% RSLogix 500 project Industrial_Bottle_Packaging_Line.RSS, saved by version 8.30.00.16 %
PROJECT "PROC1"    % processor: Bul.1763 MicroLogix 1100 Series B %

PROGRAM FILES
  LAD 2 "MAIN"  11 rungs
  LAD 3 "I / O"  27 rungs
  LAD 4 "MODE CTRL"  9 rungs
  LAD 5 "SNS IN CTR"  6 rungs
  LAD 6 "SIMULATION"  39 rungs
  LAD 7 "DEVICE CTR"  6 rungs
  LAD 8 "CYCLE RST"  2 rungs
  LAD 9 "HOURMETER"  8 rungs
  LAD 10 "ALARMS"  21 rungs

DATA FILES
  O0 OUTPUT  7 elements
  I1 INPUT  12 elements
  S2 STATUS  66 elements
  B3 BINARY  11 elements
  T4 TIMER  21 elements
  C5 COUNTER  1 elements
  R6 CONTROL  1 elements
  N7 INTEGER  23 elements
  F8 FLOAT  1 elements
  L9 LONGINT  1 elements

LADDER 2 "MAIN"
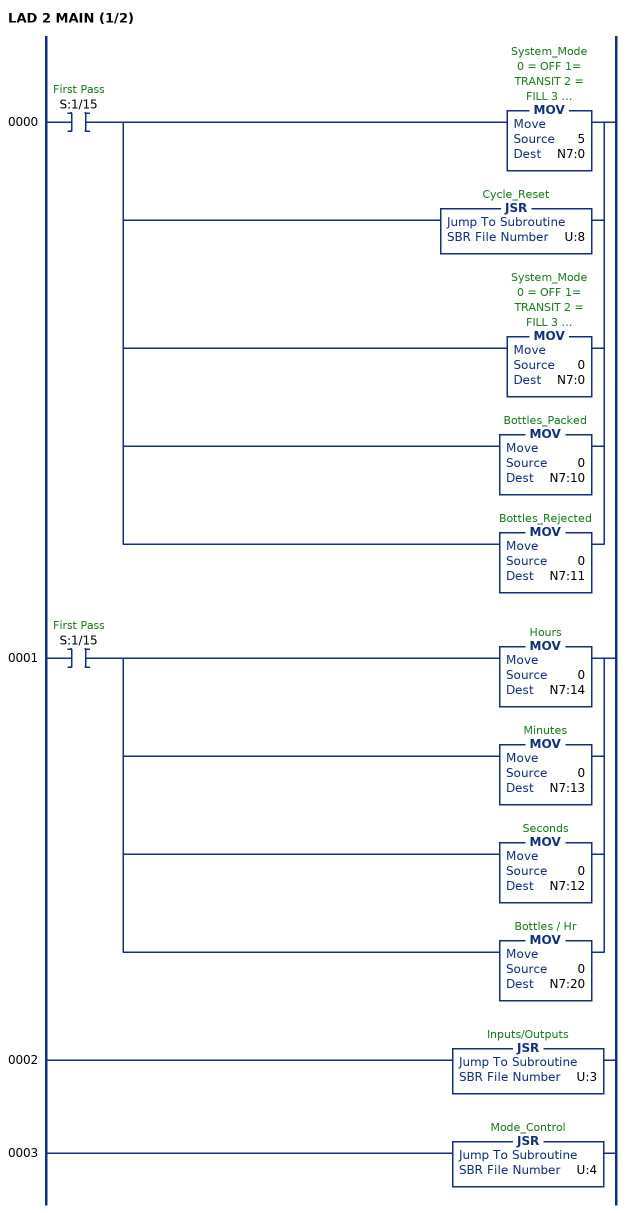
% Rung: 0 %
SOR XIC S:1/15 BST MOV 5 N7:0 NXB JSR U:8 NXB MOV 0 N7:0 NXB MOV 0 N7:10 NXB MOV 0 N7:11 BND EOR
%   S:1/15  "First Pass" %
%   N7:0  "System_Mode 0 = OFF 1= TRANSIT 2 = FILL 3 = CAPPING 4 = SORTING 5= CYC.R" %
%   U:8  "Cycle_Reset" %
%   N7:10  "Bottles_Packed" %
%   N7:11  "Bottles_Rejected" %
% Rung: 1 %
SOR XIC S:1/15 BST MOV 0 N7:14 NXB MOV 0 N7:13 NXB MOV 0 N7:12 NXB MOV 0 N7:20 BND EOR
%   S:1/15  "First Pass" %
%   N7:14  "Hours" %
%   N7:13  "Minutes" %
%   N7:12  "Seconds" %
%   N7:20  "Bottles / Hr" %
% Rung: 2 %
SOR JSR U:3 EOR
%   U:3  "Inputs/Outputs" %
% Rung: 3 %
SOR JSR U:4 EOR
%   U:4  "Mode_Control" %

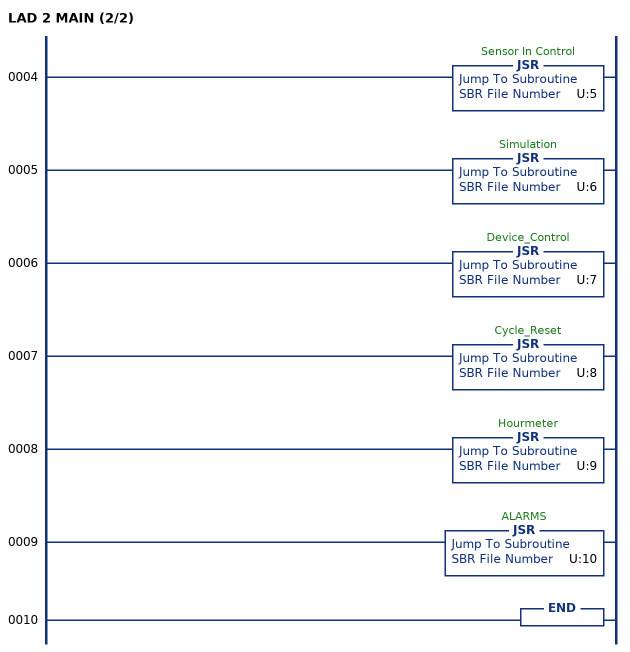
% Rung: 4 %
SOR JSR U:5 EOR
%   U:5  "Sensor In Control" %
% Rung: 5 %
SOR JSR U:6 EOR
%   U:6  "Simulation" %
% Rung: 6 %
SOR JSR U:7 EOR
%   U:7  "Device_Control" %
% Rung: 7 %
SOR JSR U:8 EOR
%   U:8  "Cycle_Reset" %
% Rung: 8 %
SOR JSR U:9 EOR
%   U:9  "Hourmeter" %
% Rung: 9 %
SOR JSR U:10 EOR
%   U:10  "ALARMS" %
% Rung: 10 %
SOR END EOR

LADDER 3 "I / O"
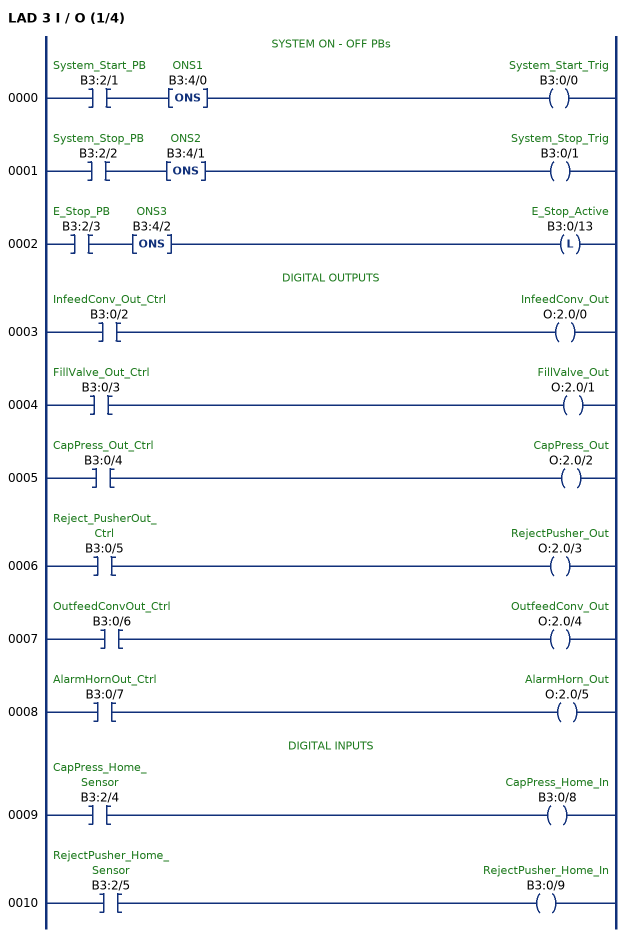
% Rung: 0 %
% SYSTEM ON - OFF PBs %
SOR XIC B3:2/1 ONS B3:4/0 OTE B3:0/0 EOR
%   B3:2/1  "System_Start_PB" %
%   B3:4/0  "ONS1" %
%   B3:0/0  "System_Start_Trig" %
% Rung: 1 %
SOR XIC B3:2/2 ONS B3:4/1 OTE B3:0/1 EOR
%   B3:2/2  "System_Stop_PB" %
%   B3:4/1  "ONS2" %
%   B3:0/1  "System_Stop_Trig" %
% Rung: 2 %
SOR XIC B3:2/3 ONS B3:4/2 OTL B3:0/13 EOR
%   B3:2/3  "E_Stop_PB" %
%   B3:4/2  "ONS3" %
%   B3:0/13  "E_Stop_Active" %
% Rung: 3 %
% DIGITAL OUTPUTS %
SOR XIC B3:0/2 OTE O:2.0/0 EOR
%   B3:0/2  "InfeedConv_Out_Ctrl" %
%   O:2.0/0  "InfeedConv_Out" %
% Rung: 4 %
SOR XIC B3:0/3 OTE O:2.0/1 EOR
%   B3:0/3  "FillValve_Out_Ctrl" %
%   O:2.0/1  "FillValve_Out" %
% Rung: 5 %
SOR XIC B3:0/4 OTE O:2.0/2 EOR
%   B3:0/4  "CapPress_Out_Ctrl" %
%   O:2.0/2  "CapPress_Out" %
% Rung: 6 %
SOR XIC B3:0/5 OTE O:2.0/3 EOR
%   B3:0/5  "Reject_PusherOut_ Ctrl" %
%   O:2.0/3  "RejectPusher_Out" %
% Rung: 7 %
SOR XIC B3:0/6 OTE O:2.0/4 EOR
%   B3:0/6  "OutfeedConvOut_Ctrl" %
%   O:2.0/4  "OutfeedConv_Out" %
% Rung: 8 %
SOR XIC B3:0/7 OTE O:2.0/5 EOR
%   B3:0/7  "AlarmHornOut_Ctrl" %
%   O:2.0/5  "AlarmHorn_Out" %
% Rung: 9 %
% DIGITAL INPUTS %
SOR XIC B3:2/4 OTE B3:0/8 EOR
%   B3:2/4  "CapPress_Home_Sensor" %
%   B3:0/8  "CapPress_Home_In" %
% Rung: 10 %
SOR XIC B3:2/5 OTE B3:0/9 EOR
%   B3:2/5  "RejectPusher_Home_ Sensor" %
%   B3:0/9  "RejectPusher_Home_In" %

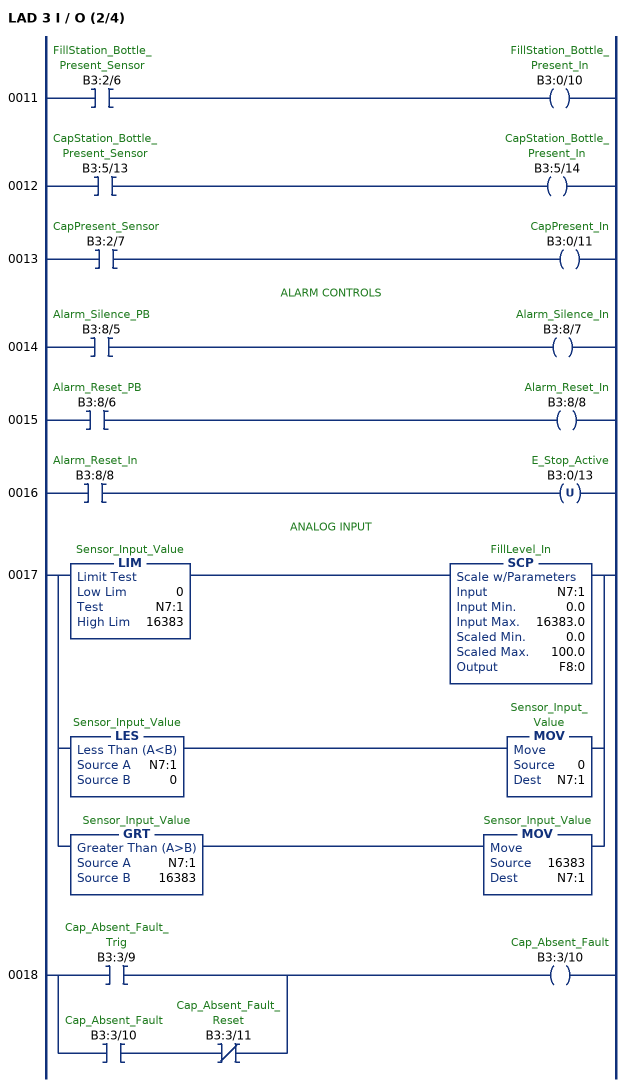
% Rung: 11 %
SOR XIC B3:2/6 OTE B3:0/10 EOR
%   B3:2/6  "FillStation_Bottle_ Present_Sensor" %
%   B3:0/10  "FillStation_Bottle_ Present_In" %
% Rung: 12 %
SOR XIC B3:5/13 OTE B3:5/14 EOR
%   B3:5/13  "CapStation_Bottle_ Present_Sensor" %
%   B3:5/14  "CapStation_Bottle_ Present_In" %
% Rung: 13 %
SOR XIC B3:2/7 OTE B3:0/11 EOR
%   B3:2/7  "CapPresent_Sensor" %
%   B3:0/11  "CapPresent_In" %
% Rung: 14 %
% ALARM CONTROLS %
SOR XIC B3:8/5 OTE B3:8/7 EOR
%   B3:8/5  "Alarm_Silence_PB" %
%   B3:8/7  "Alarm_Silence_In" %
% Rung: 15 %
SOR XIC B3:8/6 OTE B3:8/8 EOR
%   B3:8/6  "Alarm_Reset_PB" %
%   B3:8/8  "Alarm_Reset_In" %
% Rung: 16 %
SOR XIC B3:8/8 OTU B3:0/13 EOR
%   B3:8/8  "Alarm_Reset_In" %
%   B3:0/13  "E_Stop_Active" %
% Rung: 17 %
% ANALOG INPUT %
SOR BST LIM 0 N7:1 16383 SCP N7:1 0.0 16383.0 0.0 100.0 F8:0 NXB LES N7:1 0 MOV 0 N7:1 NXB GRT N7:1 16383 MOV 16383 N7:1 BND EOR
%   N7:1  "Sensor_Input_Value" %
%   F8:0  "FillLevel_In" %
% Rung: 18 %
SOR BST XIC B3:3/9 NXB XIC B3:3/10 XIO B3:3/11 BND OTE B3:3/10 EOR
%   B3:3/9  "Cap_Absent_Fault_ Trig" %
%   B3:3/10  "Cap_Absent_Fault" %
%   B3:3/11  "Cap_Absent_Fault_ Reset" %

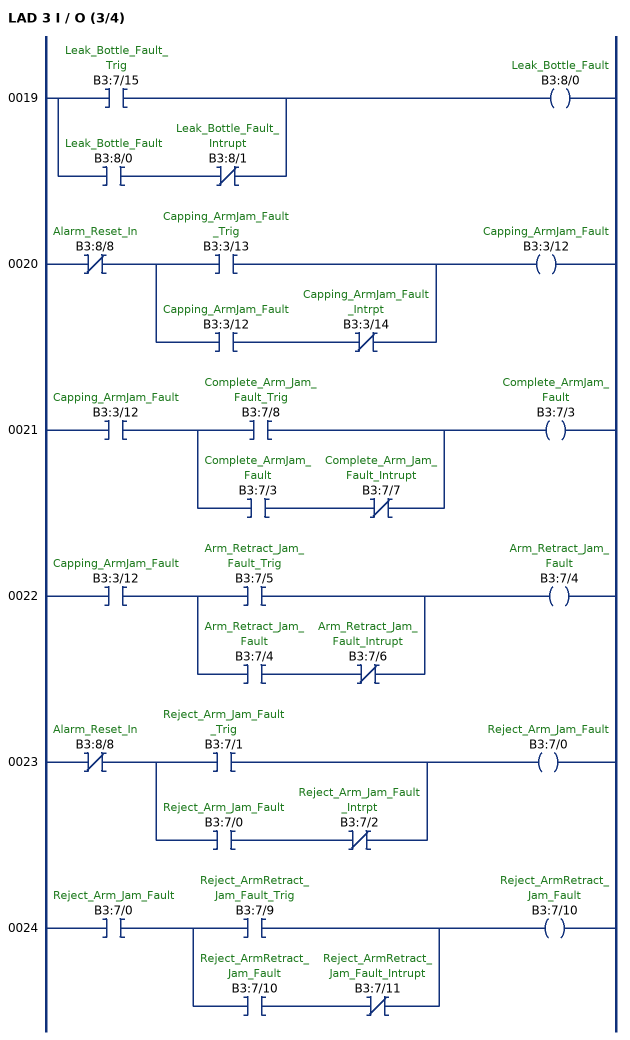
% Rung: 19 %
SOR BST XIC B3:7/15 NXB XIC B3:8/0 XIO B3:8/1 BND OTE B3:8/0 EOR
%   B3:7/15  "Leak_Bottle_Fault_ Trig" %
%   B3:8/0  "Leak_Bottle_Fault" %
%   B3:8/1  "Leak_Bottle_Fault_ Intrupt" %
% Rung: 20 %
SOR XIO B3:8/8 BST XIC B3:3/13 NXB XIC B3:3/12 XIO B3:3/14 BND OTE B3:3/12 EOR
%   B3:8/8  "Alarm_Reset_In" %
%   B3:3/13  "Capping_ArmJam_Fault _Trig" %
%   B3:3/12  "Capping_ArmJam_Fault" %
%   B3:3/14  "Capping_ArmJam_Fault _Intrpt" %
% Rung: 21 %
SOR XIC B3:3/12 BST XIC B3:7/8 NXB XIC B3:7/3 XIO B3:7/7 BND OTE B3:7/3 EOR
%   B3:3/12  "Capping_ArmJam_Fault" %
%   B3:7/8  "Complete_Arm_Jam_ Fault_Trig" %
%   B3:7/3  "Complete_ArmJam_ Fault" %
%   B3:7/7  "Complete_Arm_Jam_ Fault_Intrupt" %
% Rung: 22 %
SOR XIC B3:3/12 BST XIC B3:7/5 NXB XIC B3:7/4 XIO B3:7/6 BND OTE B3:7/4 EOR
%   B3:3/12  "Capping_ArmJam_Fault" %
%   B3:7/5  "Arm_Retract_Jam_ Fault_Trig" %
%   B3:7/4  "Arm_Retract_Jam_ Fault" %
%   B3:7/6  "Arm_Retract_Jam_ Fault_Intrupt" %
% Rung: 23 %
SOR XIO B3:8/8 BST XIC B3:7/1 NXB XIC B3:7/0 XIO B3:7/2 BND OTE B3:7/0 EOR
%   B3:8/8  "Alarm_Reset_In" %
%   B3:7/1  "Reject_Arm_Jam_Fault _Trig" %
%   B3:7/0  "Reject_Arm_Jam_Fault" %
%   B3:7/2  "Reject_Arm_Jam_Fault _Intrpt" %
% Rung: 24 %
SOR XIC B3:7/0 BST XIC B3:7/9 NXB XIC B3:7/10 XIO B3:7/11 BND OTE B3:7/10 EOR
%   B3:7/0  "Reject_Arm_Jam_Fault" %
%   B3:7/9  "Reject_ArmRetract_ Jam_Fault_Trig" %
%   B3:7/10  "Reject_ArmRetract_ Jam_Fault" %
%   B3:7/11  "Reject_ArmRetract_ Jam_Fault_Intrupt" %

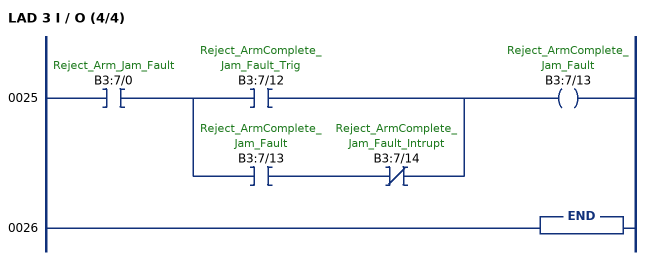
% Rung: 25 %
SOR XIC B3:7/0 BST XIC B3:7/12 NXB XIC B3:7/13 XIO B3:7/14 BND OTE B3:7/13 EOR
%   B3:7/0  "Reject_Arm_Jam_Fault" %
%   B3:7/12  "Reject_ArmComplete_ Jam_Fault_Trig" %
%   B3:7/13  "Reject_ArmComplete_ Jam_Fault" %
%   B3:7/14  "Reject_ArmComplete_ Jam_Fault_Intrupt" %
% Rung: 26 %
SOR END EOR

LADDER 4 "MODE CTRL"
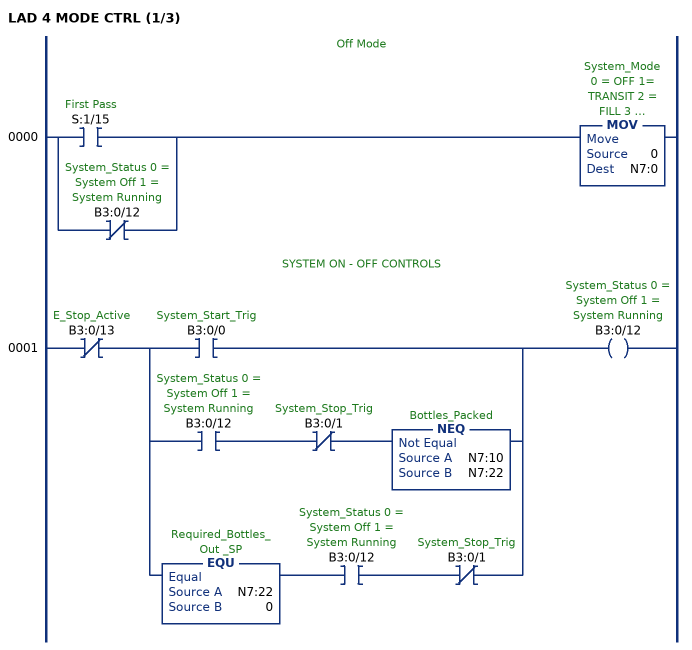
% Rung: 0 %
% Off Mode %
SOR BST XIC S:1/15 NXB XIO B3:0/12 BND MOV 0 N7:0 EOR
%   S:1/15  "First Pass" %
%   B3:0/12  "System_Status 0 = System Off 1 = System Running" %
%   N7:0  "System_Mode 0 = OFF 1= TRANSIT 2 = FILL 3 = CAPPING 4 = SORTING 5= CYC.R" %
% Rung: 1 %
% SYSTEM ON - OFF CONTROLS %
SOR XIO B3:0/13 BST XIC B3:0/0 NXB XIC B3:0/12 XIO B3:0/1 NEQ N7:10 N7:22 NXB EQU N7:22 0 XIC B3:0/12 XIO B3:0/1 BND OTE B3:0/12 EOR
%   B3:0/13  "E_Stop_Active" %
%   B3:0/0  "System_Start_Trig" %
%   B3:0/12  "System_Status 0 = System Off 1 = System Running" %
%   B3:0/1  "System_Stop_Trig" %
%   N7:10  "Bottles_Packed" %
%   N7:22  "Required_Bottles_Out _SP" %

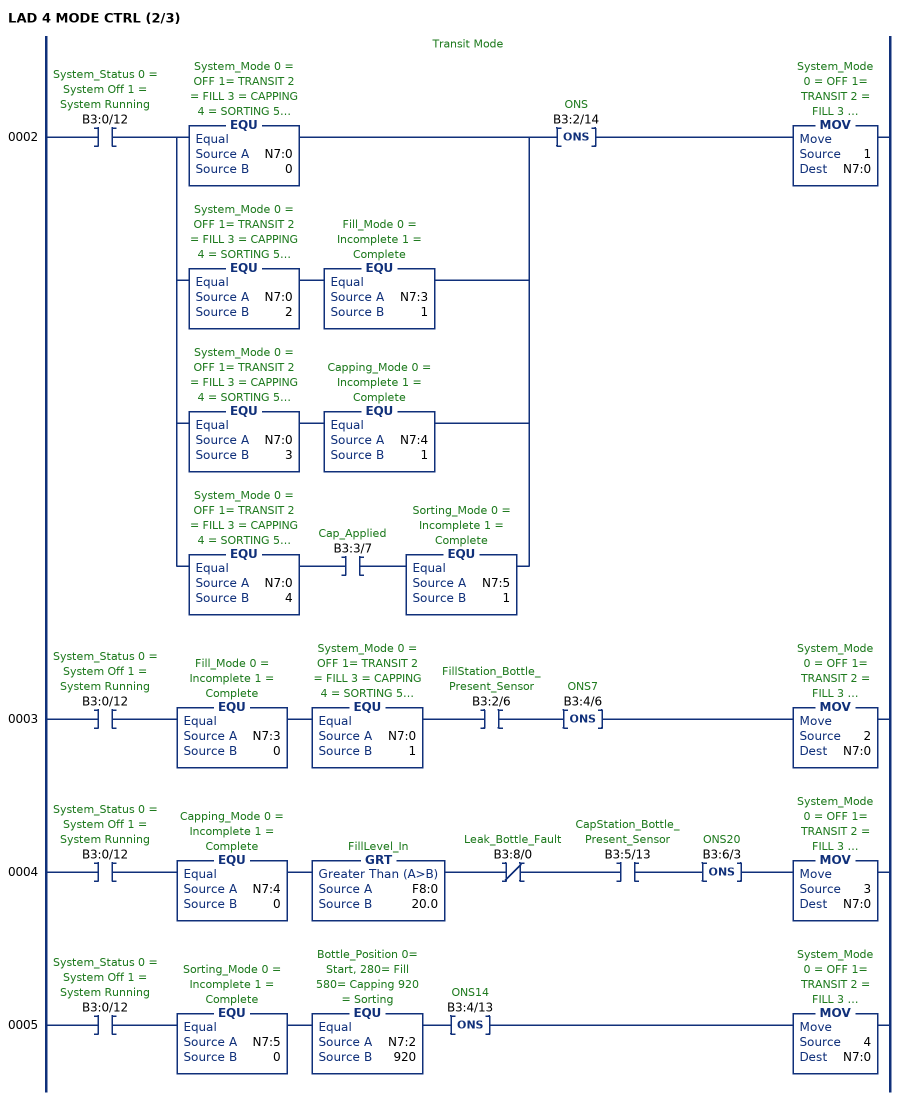
% Rung: 2 %
% Transit Mode %
SOR XIC B3:0/12 BST EQU N7:0 0 NXB EQU N7:0 2 EQU N7:3 1 NXB EQU N7:0 3 EQU N7:4 1 NXB EQU N7:0 4 XIC B3:3/7 EQU N7:5 1 BND ONS B3:2/14 MOV 1 N7:0 EOR
%   B3:0/12  "System_Status 0 = System Off 1 = System Running" %
%   N7:0  "System_Mode 0 = OFF 1= TRANSIT 2 = FILL 3 = CAPPING 4 = SORTING 5= CYC.R" %
%   N7:3  "Fill_Mode 0 = Incomplete 1 = Complete" %
%   N7:4  "Capping_Mode 0 = Incomplete 1 = Complete" %
%   B3:3/7  "Cap_Applied" %
%   N7:5  "Sorting_Mode 0 = Incomplete 1 = Complete" %
%   B3:2/14  "ONS" %
% Rung: 3 %
SOR XIC B3:0/12 EQU N7:3 0 EQU N7:0 1 XIC B3:2/6 ONS B3:4/6 MOV 2 N7:0 EOR
%   B3:0/12  "System_Status 0 = System Off 1 = System Running" %
%   N7:3  "Fill_Mode 0 = Incomplete 1 = Complete" %
%   N7:0  "System_Mode 0 = OFF 1= TRANSIT 2 = FILL 3 = CAPPING 4 = SORTING 5= CYC.R" %
%   B3:2/6  "FillStation_Bottle_ Present_Sensor" %
%   B3:4/6  "ONS7" %
% Rung: 4 %
SOR XIC B3:0/12 EQU N7:4 0 GRT F8:0 20.0 XIO B3:8/0 XIC B3:5/13 ONS B3:6/3 MOV 3 N7:0 EOR
%   B3:0/12  "System_Status 0 = System Off 1 = System Running" %
%   N7:4  "Capping_Mode 0 = Incomplete 1 = Complete" %
%   F8:0  "FillLevel_In" %
%   B3:8/0  "Leak_Bottle_Fault" %
%   B3:5/13  "CapStation_Bottle_ Present_Sensor" %
%   B3:6/3  "ONS20" %
%   N7:0  "System_Mode 0 = OFF 1= TRANSIT 2 = FILL 3 = CAPPING 4 = SORTING 5= CYC.R" %
% Rung: 5 %
SOR XIC B3:0/12 EQU N7:5 0 EQU N7:2 920 ONS B3:4/13 MOV 4 N7:0 EOR
%   B3:0/12  "System_Status 0 = System Off 1 = System Running" %
%   N7:5  "Sorting_Mode 0 = Incomplete 1 = Complete" %
%   N7:2  "Bottle_Position 0= Start, 280= Fill 580= Capping 920 = Sorting" %
%   B3:4/13  "ONS14" %
%   N7:0  "System_Mode 0 = OFF 1= TRANSIT 2 = FILL 3 = CAPPING 4 = SORTING 5= CYC.R" %

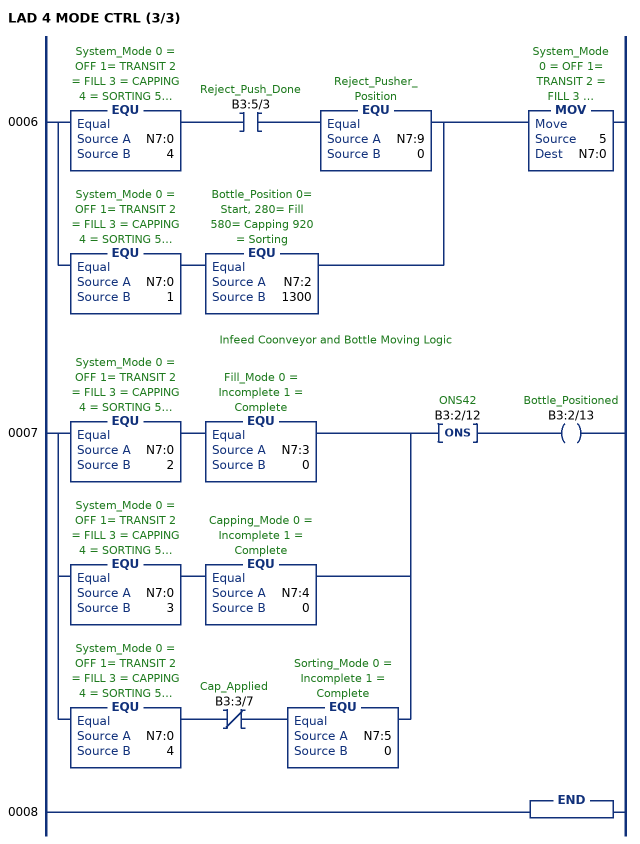
% Rung: 6 %
SOR BST EQU N7:0 4 XIC B3:5/3 EQU N7:9 0 NXB EQU N7:0 1 EQU N7:2 1300 BND MOV 5 N7:0 EOR
%   N7:0  "System_Mode 0 = OFF 1= TRANSIT 2 = FILL 3 = CAPPING 4 = SORTING 5= CYC.R" %
%   B3:5/3  "Reject_Push_Done" %
%   N7:9  "Reject_Pusher_ Position" %
%   N7:2  "Bottle_Position 0= Start, 280= Fill 580= Capping 920 = Sorting" %
% Rung: 7 %
% Infeed Coonveyor and Bottle Moving Logic %
SOR BST EQU N7:0 2 EQU N7:3 0 NXB EQU N7:0 3 EQU N7:4 0 NXB EQU N7:0 4 XIO B3:3/7 EQU N7:5 0 BND ONS B3:2/12 OTE B3:2/13 EOR
%   N7:0  "System_Mode 0 = OFF 1= TRANSIT 2 = FILL 3 = CAPPING 4 = SORTING 5= CYC.R" %
%   N7:3  "Fill_Mode 0 = Incomplete 1 = Complete" %
%   N7:4  "Capping_Mode 0 = Incomplete 1 = Complete" %
%   B3:3/7  "Cap_Applied" %
%   N7:5  "Sorting_Mode 0 = Incomplete 1 = Complete" %
%   B3:2/12  "ONS42" %
%   B3:2/13  "Bottle_Positioned" %
% Rung: 8 %
SOR END EOR

LADDER 5 "SNS IN CTR"
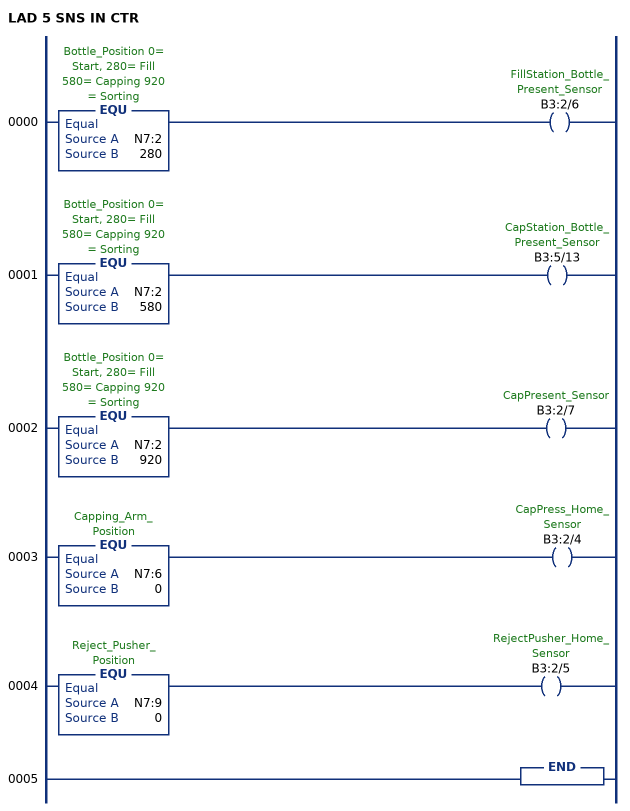
% Rung: 0 %
SOR EQU N7:2 280 OTE B3:2/6 EOR
%   N7:2  "Bottle_Position 0= Start, 280= Fill 580= Capping 920 = Sorting" %
%   B3:2/6  "FillStation_Bottle_ Present_Sensor" %
% Rung: 1 %
SOR EQU N7:2 580 OTE B3:5/13 EOR
%   N7:2  "Bottle_Position 0= Start, 280= Fill 580= Capping 920 = Sorting" %
%   B3:5/13  "CapStation_Bottle_ Present_Sensor" %
% Rung: 2 %
SOR EQU N7:2 920 OTE B3:2/7 EOR
%   N7:2  "Bottle_Position 0= Start, 280= Fill 580= Capping 920 = Sorting" %
%   B3:2/7  "CapPresent_Sensor" %
% Rung: 3 %
SOR EQU N7:6 0 OTE B3:2/4 EOR
%   N7:6  "Capping_Arm_Position" %
%   B3:2/4  "CapPress_Home_Sensor" %
% Rung: 4 %
SOR EQU N7:9 0 OTE B3:2/5 EOR
%   N7:9  "Reject_Pusher_ Position" %
%   B3:2/5  "RejectPusher_Home_ Sensor" %
% Rung: 5 %
SOR END EOR

LADDER 6 "SIMULATION"
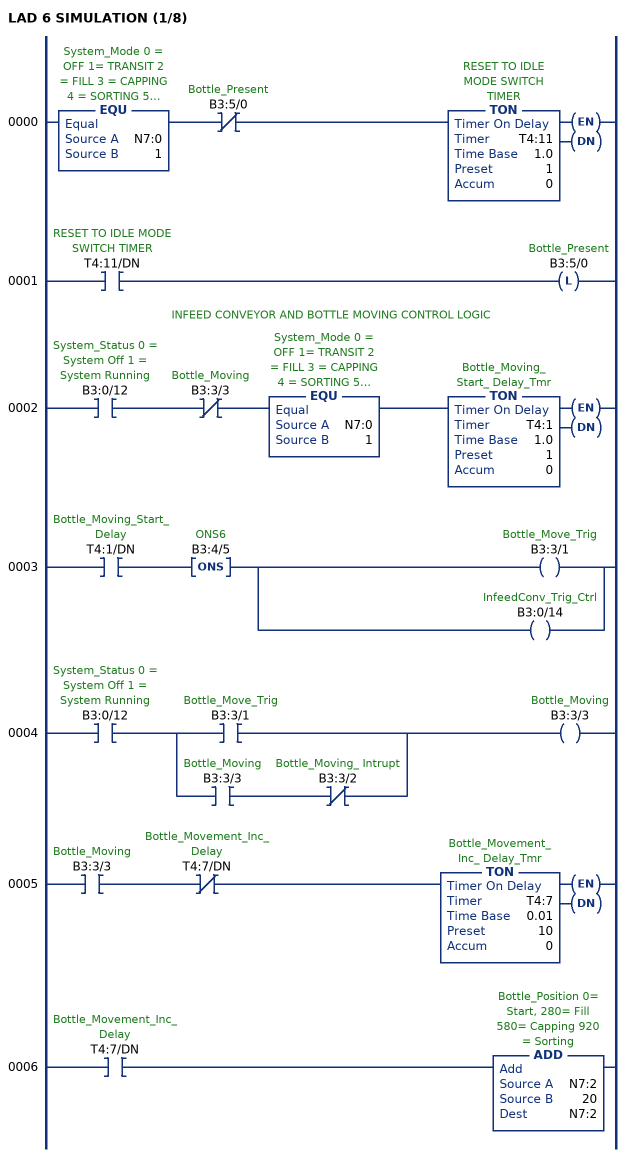
% Rung: 0 %
SOR EQU N7:0 1 XIO B3:5/0 TON T4:11 1.0 1 0 EOR
%   N7:0  "System_Mode 0 = OFF 1= TRANSIT 2 = FILL 3 = CAPPING 4 = SORTING 5= CYC.R" %
%   B3:5/0  "Bottle_Present" %
%   T4:11  "RESET TO IDLE MODE SWITCH TIMER" %
% Rung: 1 %
SOR XIC T4:11/DN OTL B3:5/0 EOR
%   T4:11  "RESET TO IDLE MODE SWITCH TIMER" %
%   B3:5/0  "Bottle_Present" %
% Rung: 2 %
% INFEED CONVEYOR AND BOTTLE MOVING CONTROL LOGIC %
SOR XIC B3:0/12 XIO B3:3/3 EQU N7:0 1 TON T4:1 1.0 1 0 EOR
%   B3:0/12  "System_Status 0 = System Off 1 = System Running" %
%   B3:3/3  "Bottle_Moving" %
%   N7:0  "System_Mode 0 = OFF 1= TRANSIT 2 = FILL 3 = CAPPING 4 = SORTING 5= CYC.R" %
%   T4:1  "Bottle_Moving_Start_ Delay_Tmr" %
% Rung: 3 %
SOR XIC T4:1/DN ONS B3:4/5 BST OTE B3:3/1 NXB OTE B3:0/14 BND EOR
%   T4:1/DN  "Bottle_Moving_Start_ Delay" %
%   B3:4/5  "ONS6" %
%   B3:3/1  "Bottle_Move_Trig" %
%   B3:0/14  "InfeedConv_Trig_Ctrl" %
% Rung: 4 %
SOR XIC B3:0/12 BST XIC B3:3/1 NXB XIC B3:3/3 XIO B3:3/2 BND OTE B3:3/3 EOR
%   B3:0/12  "System_Status 0 = System Off 1 = System Running" %
%   B3:3/1  "Bottle_Move_Trig" %
%   B3:3/3  "Bottle_Moving" %
%   B3:3/2  "Bottle_Moving_ Intrupt" %
% Rung: 5 %
SOR XIC B3:3/3 XIO T4:7/DN TON T4:7 0.01 10 0 EOR
%   B3:3/3  "Bottle_Moving" %
%   T4:7/DN  "Bottle_Movement_Inc_ Delay" %
%   T4:7  "Bottle_Movement_Inc_ Delay_Tmr" %
% Rung: 6 %
SOR XIC T4:7/DN ADD N7:2 20 N7:2 EOR
%   T4:7/DN  "Bottle_Movement_Inc_ Delay" %
%   N7:2  "Bottle_Position 0= Start, 280= Fill 580= Capping 920 = Sorting" %

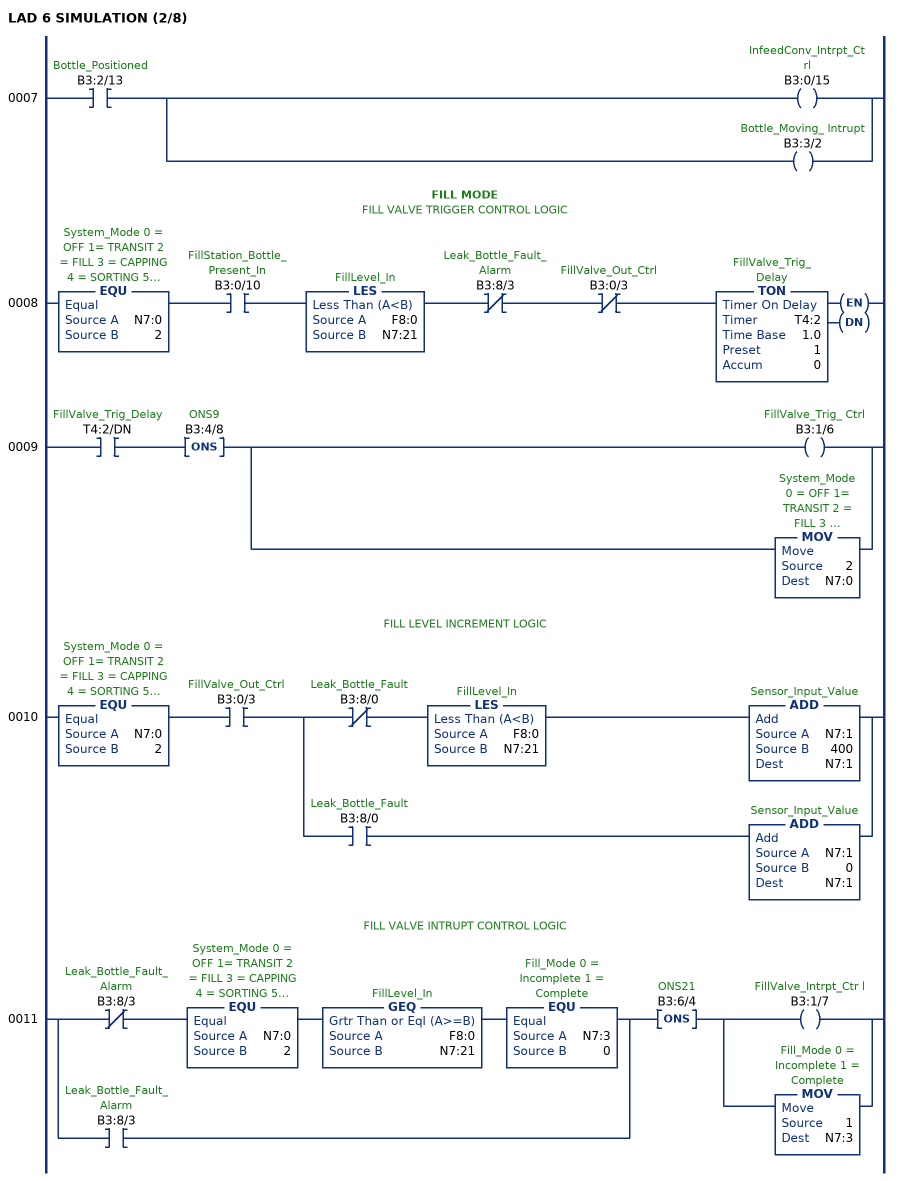
% Rung: 7 %
SOR XIC B3:2/13 BST OTE B3:0/15 NXB OTE B3:3/2 BND EOR
%   B3:2/13  "Bottle_Positioned" %
%   B3:0/15  "InfeedConv_Intrpt_Ct rl" %
%   B3:3/2  "Bottle_Moving_ Intrupt" %
% Rung: 8 %
% TITLE: FILL MODE %
% FILL VALVE TRIGGER CONTROL LOGIC %
SOR EQU N7:0 2 XIC B3:0/10 LES F8:0 N7:21 XIO B3:8/3 XIO B3:0/3 TON T4:2 1.0 1 0 EOR
%   N7:0  "System_Mode 0 = OFF 1= TRANSIT 2 = FILL 3 = CAPPING 4 = SORTING 5= CYC.R" %
%   B3:0/10  "FillStation_Bottle_ Present_In" %
%   F8:0  "FillLevel_In" %
%   N7:21  "Fill_LVL_SP" %
%   B3:8/3  "Leak_Bottle_Fault_ Alarm" %
%   B3:0/3  "FillValve_Out_Ctrl" %
%   T4:2  "FillValve_Trig_ Delay" %
% Rung: 9 %
SOR XIC T4:2/DN ONS B3:4/8 BST OTE B3:1/6 NXB MOV 2 N7:0 BND EOR
%   T4:2/DN  "FillValve_Trig_Delay" %
%   B3:4/8  "ONS9" %
%   B3:1/6  "FillValve_Trig_ Ctrl" %
%   N7:0  "System_Mode 0 = OFF 1= TRANSIT 2 = FILL 3 = CAPPING 4 = SORTING 5= CYC.R" %
% Rung: 10 %
% FILL LEVEL INCREMENT LOGIC %
SOR EQU N7:0 2 XIC B3:0/3 BST XIO B3:8/0 LES F8:0 N7:21 ADD N7:1 400 N7:1 NXB XIC B3:8/0 ADD N7:1 0 N7:1 BND EOR
%   N7:0  "System_Mode 0 = OFF 1= TRANSIT 2 = FILL 3 = CAPPING 4 = SORTING 5= CYC.R" %
%   B3:0/3  "FillValve_Out_Ctrl" %
%   B3:8/0  "Leak_Bottle_Fault" %
%   F8:0  "FillLevel_In" %
%   N7:21  "Fill_LVL_SP" %
%   N7:1  "Sensor_Input_Value" %
% Rung: 11 %
% FILL VALVE INTRUPT CONTROL LOGIC %
SOR BST XIO B3:8/3 EQU N7:0 2 GEQ F8:0 N7:21 EQU N7:3 0 NXB XIC B3:8/3 BND ONS B3:6/4 BST OTE B3:1/7 NXB MOV 1 N7:3 BND EOR
%   B3:8/3  "Leak_Bottle_Fault_ Alarm" %
%   N7:0  "System_Mode 0 = OFF 1= TRANSIT 2 = FILL 3 = CAPPING 4 = SORTING 5= CYC.R" %
%   F8:0  "FillLevel_In" %
%   N7:21  "Fill_LVL_SP" %
%   N7:3  "Fill_Mode 0 = Incomplete 1 = Complete" %
%   B3:6/4  "ONS21" %
%   B3:1/7  "FillValve_Intrpt_Ctr l" %

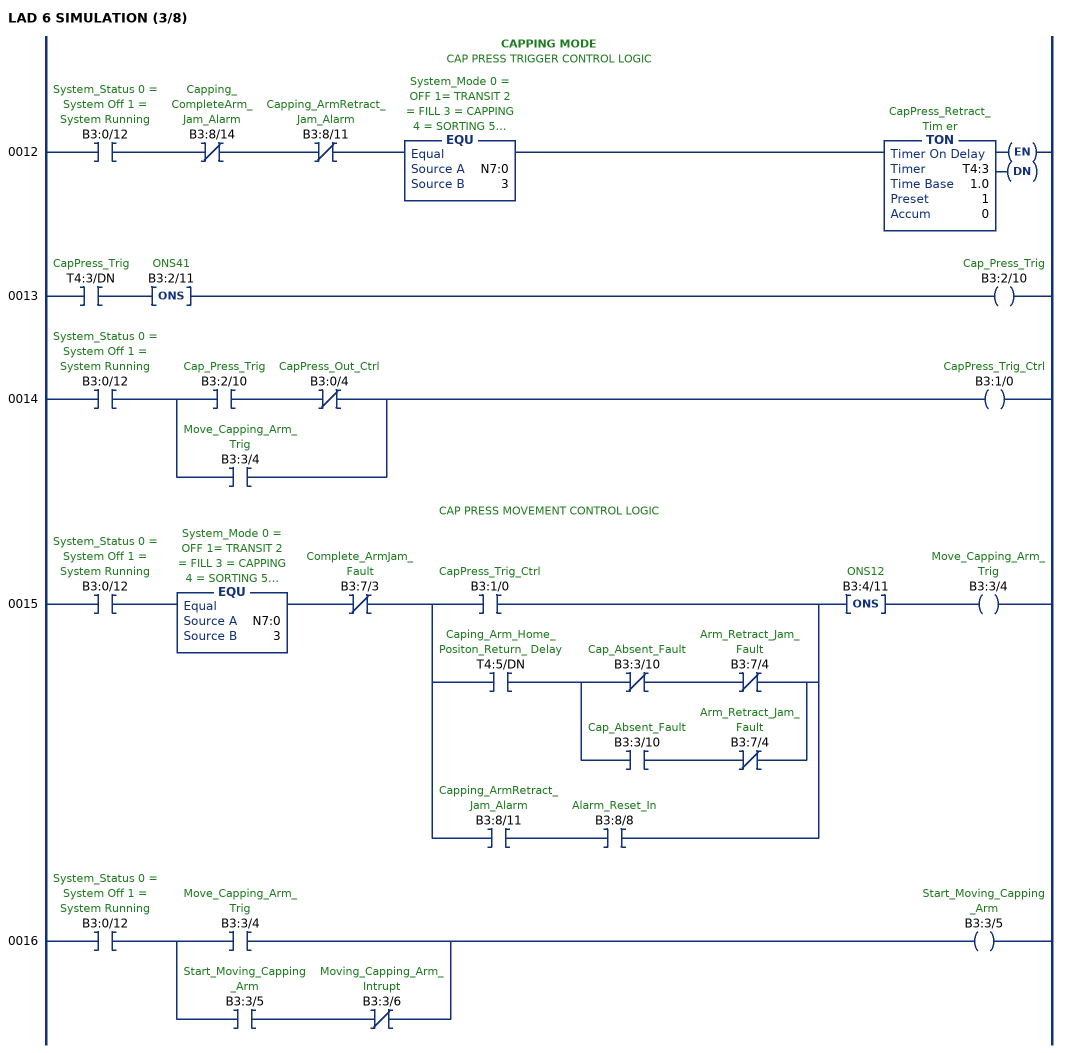
% Rung: 12 %
% TITLE: CAPPING MODE %
% CAP PRESS TRIGGER CONTROL LOGIC %
SOR XIC B3:0/12 XIO B3:8/14 XIO B3:8/11 EQU N7:0 3 TON T4:3 1.0 1 0 EOR
%   B3:0/12  "System_Status 0 = System Off 1 = System Running" %
%   B3:8/14  "Capping_CompleteArm_ Jam_Alarm" %
%   B3:8/11  "Capping_ArmRetract_ Jam_Alarm" %
%   N7:0  "System_Mode 0 = OFF 1= TRANSIT 2 = FILL 3 = CAPPING 4 = SORTING 5= CYC.R" %
%   T4:3  "CapPress_Retract_Tim er" %
% Rung: 13 %
SOR XIC T4:3/DN ONS B3:2/11 OTE B3:2/10 EOR
%   T4:3/DN  "CapPress_Trig" %
%   B3:2/11  "ONS41" %
%   B3:2/10  "Cap_Press_Trig" %
% Rung: 14 %
SOR XIC B3:0/12 BST XIC B3:2/10 XIO B3:0/4 NXB XIC B3:3/4 BND OTE B3:1/0 EOR
%   B3:0/12  "System_Status 0 = System Off 1 = System Running" %
%   B3:2/10  "Cap_Press_Trig" %
%   B3:0/4  "CapPress_Out_Ctrl" %
%   B3:3/4  "Move_Capping_Arm_ Trig" %
%   B3:1/0  "CapPress_Trig_Ctrl" %
% Rung: 15 %
% CAP PRESS MOVEMENT CONTROL LOGIC %
SOR XIC B3:0/12 EQU N7:0 3 XIO B3:7/3 BST XIC B3:1/0 NXB XIC T4:5/DN BST XIO B3:3/10 XIO B3:7/4 NXB XIC B3:3/10 XIO B3:7/4 BND NXB XIC B3:8/11 XIC B3:8/8 BND ONS B3:4/11 OTE B3:3/4 EOR
%   B3:0/12  "System_Status 0 = System Off 1 = System Running" %
%   N7:0  "System_Mode 0 = OFF 1= TRANSIT 2 = FILL 3 = CAPPING 4 = SORTING 5= CYC.R" %
%   B3:7/3  "Complete_ArmJam_ Fault" %
%   B3:1/0  "CapPress_Trig_Ctrl" %
%   T4:5/DN  "Caping_Arm_Home_ Positon_Return_ Delay" %
%   B3:3/10  "Cap_Absent_Fault" %
%   B3:7/4  "Arm_Retract_Jam_ Fault" %
%   B3:8/11  "Capping_ArmRetract_ Jam_Alarm" %
%   B3:8/8  "Alarm_Reset_In" %
%   B3:4/11  "ONS12" %
%   B3:3/4  "Move_Capping_Arm_ Trig" %
% Rung: 16 %
SOR XIC B3:0/12 BST XIC B3:3/4 NXB XIC B3:3/5 XIO B3:3/6 BND OTE B3:3/5 EOR
%   B3:0/12  "System_Status 0 = System Off 1 = System Running" %
%   B3:3/4  "Move_Capping_Arm_ Trig" %
%   B3:3/5  "Start_Moving_Capping _Arm" %
%   B3:3/6  "Moving_Capping_Arm_ Intrupt" %

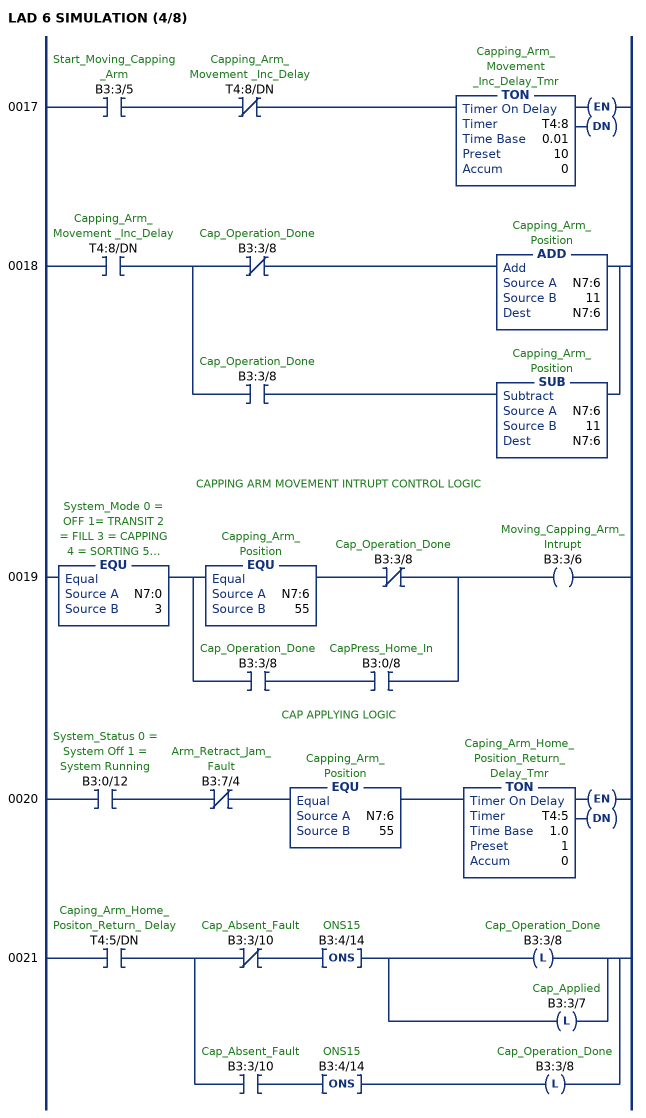
% Rung: 17 %
SOR XIC B3:3/5 XIO T4:8/DN TON T4:8 0.01 10 0 EOR
%   B3:3/5  "Start_Moving_Capping _Arm" %
%   T4:8/DN  "Capping_Arm_Movement _Inc_Delay" %
%   T4:8  "Capping_Arm_Movement _Inc_Delay_Tmr" %
% Rung: 18 %
SOR XIC T4:8/DN BST XIO B3:3/8 ADD N7:6 11 N7:6 NXB XIC B3:3/8 SUB N7:6 11 N7:6 BND EOR
%   T4:8/DN  "Capping_Arm_Movement _Inc_Delay" %
%   B3:3/8  "Cap_Operation_Done" %
%   N7:6  "Capping_Arm_Position" %
% Rung: 19 %
% CAPPING ARM MOVEMENT INTRUPT CONTROL LOGIC %
SOR EQU N7:0 3 BST EQU N7:6 55 XIO B3:3/8 NXB XIC B3:3/8 XIC B3:0/8 BND OTE B3:3/6 EOR
%   N7:0  "System_Mode 0 = OFF 1= TRANSIT 2 = FILL 3 = CAPPING 4 = SORTING 5= CYC.R" %
%   N7:6  "Capping_Arm_Position" %
%   B3:3/8  "Cap_Operation_Done" %
%   B3:0/8  "CapPress_Home_In" %
%   B3:3/6  "Moving_Capping_Arm_ Intrupt" %
% Rung: 20 %
% CAP APPLYING LOGIC %
SOR XIC B3:0/12 XIO B3:7/4 EQU N7:6 55 TON T4:5 1.0 1 0 EOR
%   B3:0/12  "System_Status 0 = System Off 1 = System Running" %
%   B3:7/4  "Arm_Retract_Jam_ Fault" %
%   N7:6  "Capping_Arm_Position" %
%   T4:5  "Caping_Arm_Home_ Position_Return_ Delay_Tmr" %
% Rung: 21 %
SOR XIC T4:5/DN BST XIO B3:3/10 ONS B3:4/14 BST OTL B3:3/8 NXB OTL B3:3/7 BND NXB XIC B3:3/10 ONS B3:4/14 OTL B3:3/8 BND EOR
%   T4:5/DN  "Caping_Arm_Home_ Positon_Return_ Delay" %
%   B3:3/10  "Cap_Absent_Fault" %
%   B3:4/14  "ONS15" %
%   B3:3/8  "Cap_Operation_Done" %
%   B3:3/7  "Cap_Applied" %

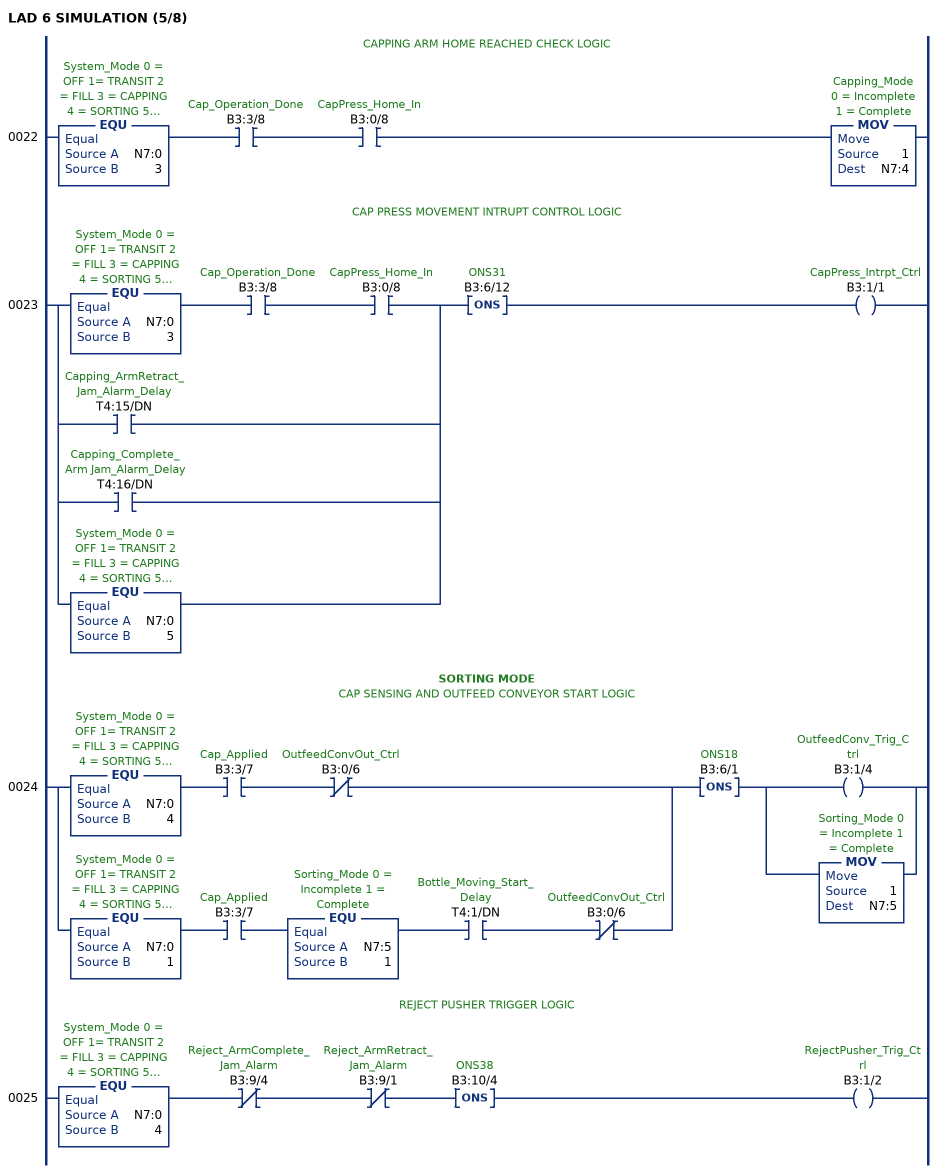
% Rung: 22 %
% CAPPING ARM HOME REACHED CHECK LOGIC %
SOR EQU N7:0 3 XIC B3:3/8 XIC B3:0/8 MOV 1 N7:4 EOR
%   N7:0  "System_Mode 0 = OFF 1= TRANSIT 2 = FILL 3 = CAPPING 4 = SORTING 5= CYC.R" %
%   B3:3/8  "Cap_Operation_Done" %
%   B3:0/8  "CapPress_Home_In" %
%   N7:4  "Capping_Mode 0 = Incomplete 1 = Complete" %
% Rung: 23 %
% CAP PRESS MOVEMENT INTRUPT CONTROL LOGIC %
SOR BST EQU N7:0 3 XIC B3:3/8 XIC B3:0/8 NXB XIC T4:15/DN NXB XIC T4:16/DN NXB EQU N7:0 5 BND ONS B3:6/12 OTE B3:1/1 EOR
%   N7:0  "System_Mode 0 = OFF 1= TRANSIT 2 = FILL 3 = CAPPING 4 = SORTING 5= CYC.R" %
%   B3:3/8  "Cap_Operation_Done" %
%   B3:0/8  "CapPress_Home_In" %
%   T4:15/DN  "Capping_ArmRetract_ Jam_Alarm_Delay" %
%   T4:16/DN  "Capping_Complete_Arm Jam_Alarm_Delay" %
%   B3:6/12  "ONS31" %
%   B3:1/1  "CapPress_Intrpt_Ctrl" %
% Rung: 24 %
% TITLE: SORTING MODE %
% CAP SENSING AND OUTFEED CONVEYOR START LOGIC %
SOR BST EQU N7:0 4 XIC B3:3/7 XIO B3:0/6 NXB EQU N7:0 1 XIC B3:3/7 EQU N7:5 1 XIC T4:1/DN XIO B3:0/6 BND ONS B3:6/1 BST OTE B3:1/4 NXB MOV 1 N7:5 BND EOR
%   N7:0  "System_Mode 0 = OFF 1= TRANSIT 2 = FILL 3 = CAPPING 4 = SORTING 5= CYC.R" %
%   B3:3/7  "Cap_Applied" %
%   B3:0/6  "OutfeedConvOut_Ctrl" %
%   N7:5  "Sorting_Mode 0 = Incomplete 1 = Complete" %
%   T4:1/DN  "Bottle_Moving_Start_ Delay" %
%   B3:6/1  "ONS18" %
%   B3:1/4  "OutfeedConv_Trig_C trl" %
% Rung: 25 %
% REJECT PUSHER TRIGGER LOGIC %
SOR EQU N7:0 4 XIO B3:9/4 XIO B3:9/1 ONS B3:10/4 OTE B3:1/2 EOR
%   N7:0  "System_Mode 0 = OFF 1= TRANSIT 2 = FILL 3 = CAPPING 4 = SORTING 5= CYC.R" %
%   B3:9/4  "Reject_ArmComplete_ Jam_Alarm" %
%   B3:9/1  "Reject_ArmRetract_ Jam_Alarm" %
%   B3:10/4  "ONS38" %
%   B3:1/2  "RejectPusher_Trig_Ct rl" %

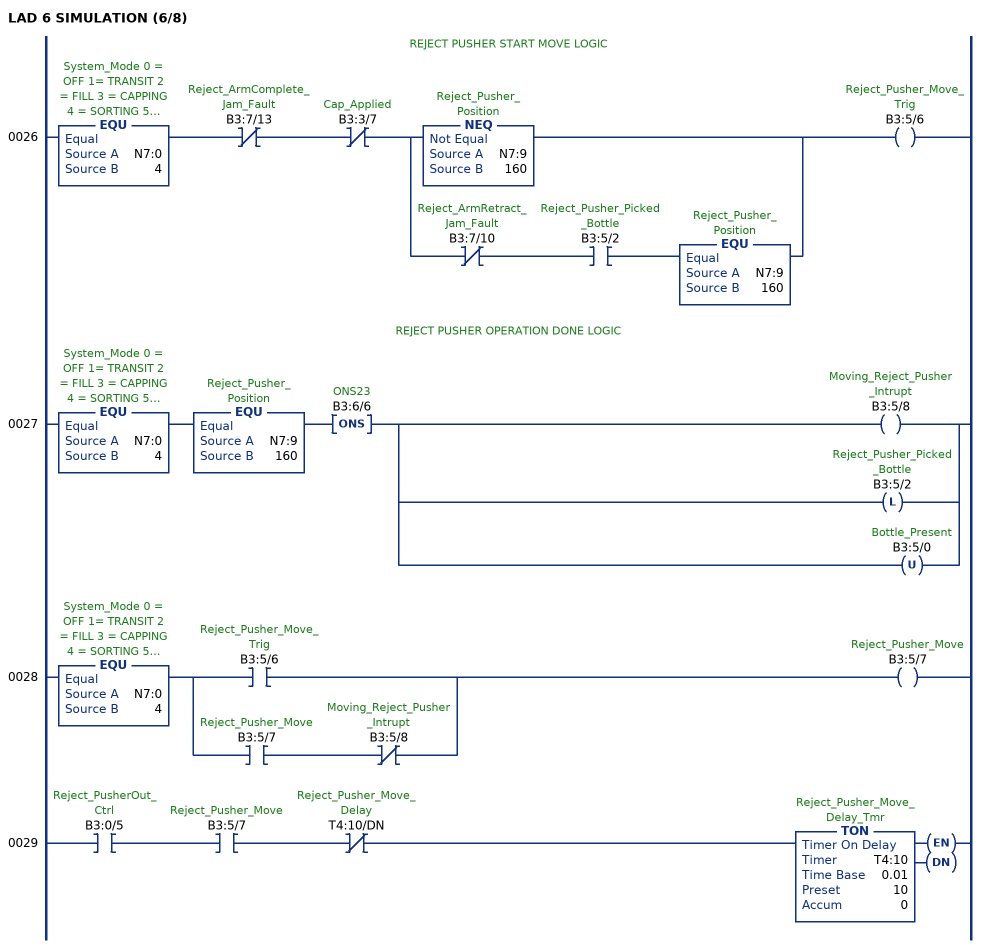
% Rung: 26 %
% REJECT PUSHER START MOVE LOGIC %
SOR EQU N7:0 4 XIO B3:7/13 XIO B3:3/7 BST NEQ N7:9 160 NXB XIO B3:7/10 XIC B3:5/2 EQU N7:9 160 BND OTE B3:5/6 EOR
%   N7:0  "System_Mode 0 = OFF 1= TRANSIT 2 = FILL 3 = CAPPING 4 = SORTING 5= CYC.R" %
%   B3:7/13  "Reject_ArmComplete_ Jam_Fault" %
%   B3:3/7  "Cap_Applied" %
%   N7:9  "Reject_Pusher_ Position" %
%   B3:7/10  "Reject_ArmRetract_ Jam_Fault" %
%   B3:5/2  "Reject_Pusher_Picked _Bottle" %
%   B3:5/6  "Reject_Pusher_Move_ Trig" %
% Rung: 27 %
% REJECT PUSHER OPERATION DONE LOGIC %
SOR EQU N7:0 4 EQU N7:9 160 ONS B3:6/6 BST OTE B3:5/8 NXB OTL B3:5/2 NXB OTU B3:5/0 BND EOR
%   N7:0  "System_Mode 0 = OFF 1= TRANSIT 2 = FILL 3 = CAPPING 4 = SORTING 5= CYC.R" %
%   N7:9  "Reject_Pusher_ Position" %
%   B3:6/6  "ONS23" %
%   B3:5/8  "Moving_Reject_Pusher _Intrupt" %
%   B3:5/2  "Reject_Pusher_Picked _Bottle" %
%   B3:5/0  "Bottle_Present" %
% Rung: 28 %
SOR EQU N7:0 4 BST XIC B3:5/6 NXB XIC B3:5/7 XIO B3:5/8 BND OTE B3:5/7 EOR
%   N7:0  "System_Mode 0 = OFF 1= TRANSIT 2 = FILL 3 = CAPPING 4 = SORTING 5= CYC.R" %
%   B3:5/6  "Reject_Pusher_Move_ Trig" %
%   B3:5/7  "Reject_Pusher_Move" %
%   B3:5/8  "Moving_Reject_Pusher _Intrupt" %
% Rung: 29 %
SOR XIC B3:0/5 XIC B3:5/7 XIO T4:10/DN TON T4:10 0.01 10 0 EOR
%   B3:0/5  "Reject_PusherOut_ Ctrl" %
%   B3:5/7  "Reject_Pusher_Move" %
%   T4:10/DN  "Reject_Pusher_Move_ Delay" %
%   T4:10  "Reject_Pusher_Move_ Delay_Tmr" %

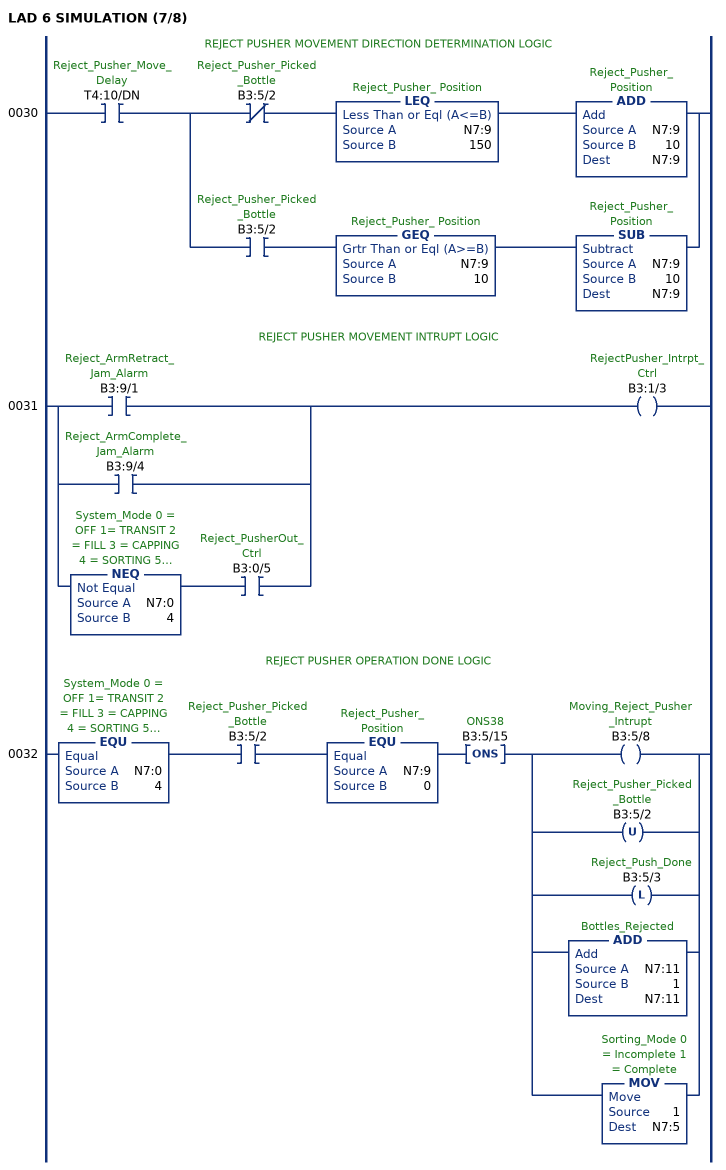
% Rung: 30 %
% REJECT PUSHER MOVEMENT DIRECTION DETERMINATION LOGIC %
SOR XIC T4:10/DN BST XIO B3:5/2 LEQ N7:9 150 ADD N7:9 10 N7:9 NXB XIC B3:5/2 GEQ N7:9 10 SUB N7:9 10 N7:9 BND EOR
%   T4:10/DN  "Reject_Pusher_Move_ Delay" %
%   B3:5/2  "Reject_Pusher_Picked _Bottle" %
%   N7:9  "Reject_Pusher_ Position" %
% Rung: 31 %
% REJECT PUSHER MOVEMENT INTRUPT LOGIC %
SOR BST XIC B3:9/1 NXB XIC B3:9/4 NXB NEQ N7:0 4 XIC B3:0/5 BND OTE B3:1/3 EOR
%   B3:9/1  "Reject_ArmRetract_ Jam_Alarm" %
%   B3:9/4  "Reject_ArmComplete_ Jam_Alarm" %
%   N7:0  "System_Mode 0 = OFF 1= TRANSIT 2 = FILL 3 = CAPPING 4 = SORTING 5= CYC.R" %
%   B3:0/5  "Reject_PusherOut_ Ctrl" %
%   B3:1/3  "RejectPusher_Intrpt_ Ctrl" %
% Rung: 32 %
% REJECT PUSHER OPERATION DONE LOGIC %
SOR EQU N7:0 4 XIC B3:5/2 EQU N7:9 0 ONS B3:5/15 BST OTE B3:5/8 NXB OTU B3:5/2 NXB OTL B3:5/3 NXB ADD N7:11 1 N7:11 NXB MOV 1 N7:5 BND EOR
%   N7:0  "System_Mode 0 = OFF 1= TRANSIT 2 = FILL 3 = CAPPING 4 = SORTING 5= CYC.R" %
%   B3:5/2  "Reject_Pusher_Picked _Bottle" %
%   N7:9  "Reject_Pusher_ Position" %
%   B3:5/15  "ONS38" %
%   B3:5/8  "Moving_Reject_Pusher _Intrupt" %
%   B3:5/3  "Reject_Push_Done" %
%   N7:11  "Bottles_Rejected" %
%   N7:5  "Sorting_Mode 0 = Incomplete 1 = Complete" %

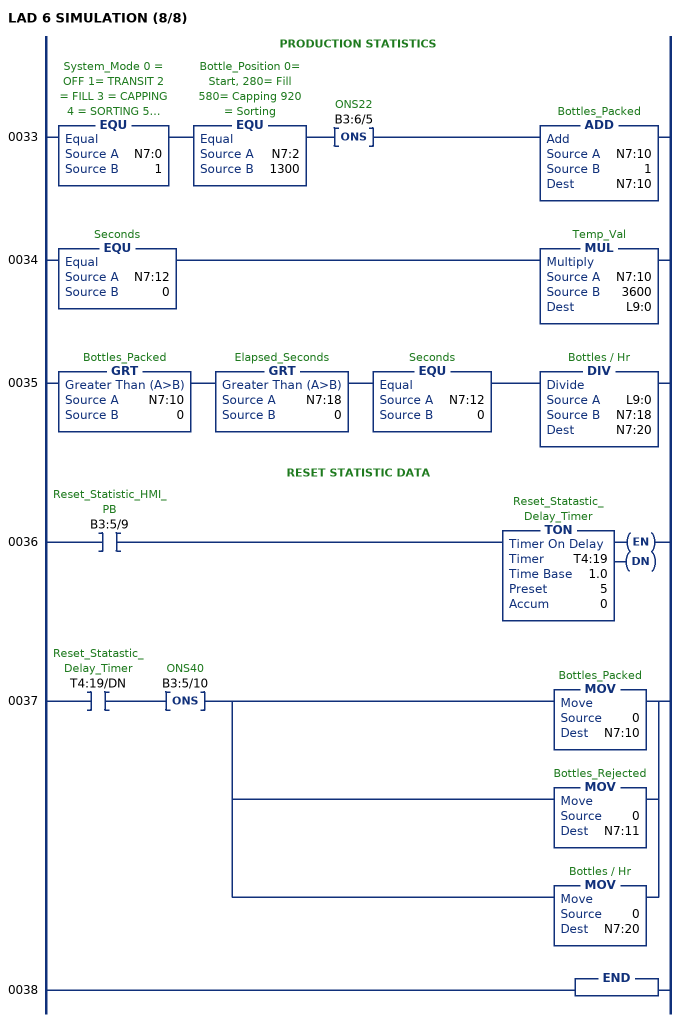
% Rung: 33 %
% TITLE: PRODUCTION STATISTICS %
SOR EQU N7:0 1 EQU N7:2 1300 ONS B3:6/5 ADD N7:10 1 N7:10 EOR
%   N7:0  "System_Mode 0 = OFF 1= TRANSIT 2 = FILL 3 = CAPPING 4 = SORTING 5= CYC.R" %
%   N7:2  "Bottle_Position 0= Start, 280= Fill 580= Capping 920 = Sorting" %
%   B3:6/5  "ONS22" %
%   N7:10  "Bottles_Packed" %
% Rung: 34 %
SOR EQU N7:12 0 MUL N7:10 3600 L9:0 EOR
%   N7:12  "Seconds" %
%   N7:10  "Bottles_Packed" %
%   L9:0  "Temp_Val" %
% Rung: 35 %
SOR GRT N7:10 0 GRT N7:18 0 EQU N7:12 0 DIV L9:0 N7:18 N7:20 EOR
%   N7:10  "Bottles_Packed" %
%   N7:18  "Elapsed_Seconds" %
%   N7:12  "Seconds" %
%   L9:0  "Temp_Val" %
%   N7:20  "Bottles / Hr" %
% Rung: 36 %
% TITLE: RESET STATISTIC DATA %
SOR XIC B3:5/9 TON T4:19 1.0 5 0 EOR
%   B3:5/9  "Reset_Statistic_HMI_ PB" %
%   T4:19  "Reset_Statastic_ Delay_Timer" %
% Rung: 37 %
SOR XIC T4:19/DN ONS B3:5/10 BST MOV 0 N7:10 NXB MOV 0 N7:11 NXB MOV 0 N7:20 BND EOR
%   T4:19  "Reset_Statastic_ Delay_Timer" %
%   B3:5/10  "ONS40" %
%   N7:10  "Bottles_Packed" %
%   N7:11  "Bottles_Rejected" %
%   N7:20  "Bottles / Hr" %
% Rung: 38 %
SOR END EOR

LADDER 7 "DEVICE CTR"
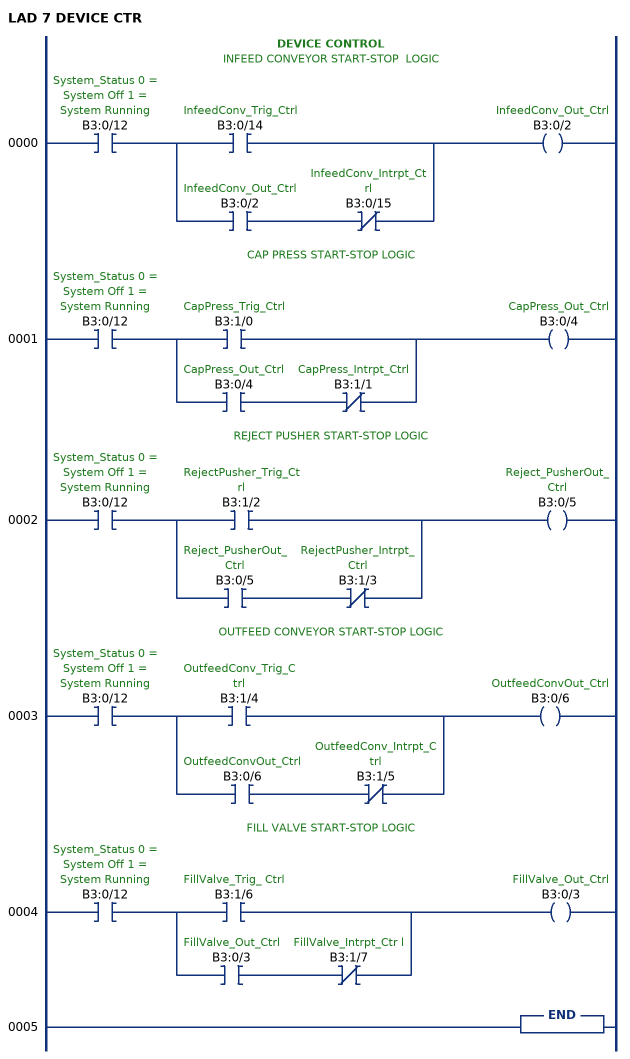
% Rung: 0 %
% TITLE: DEVICE CONTROL %
% INFEED CONVEYOR START-STOP  LOGIC %
SOR XIC B3:0/12 BST XIC B3:0/14 NXB XIC B3:0/2 XIO B3:0/15 BND OTE B3:0/2 EOR
%   B3:0/12  "System_Status 0 = System Off 1 = System Running" %
%   B3:0/14  "InfeedConv_Trig_Ctrl" %
%   B3:0/2  "InfeedConv_Out_Ctrl" %
%   B3:0/15  "InfeedConv_Intrpt_Ct rl" %
% Rung: 1 %
% CAP PRESS START-STOP LOGIC %
SOR XIC B3:0/12 BST XIC B3:1/0 NXB XIC B3:0/4 XIO B3:1/1 BND OTE B3:0/4 EOR
%   B3:0/12  "System_Status 0 = System Off 1 = System Running" %
%   B3:1/0  "CapPress_Trig_Ctrl" %
%   B3:0/4  "CapPress_Out_Ctrl" %
%   B3:1/1  "CapPress_Intrpt_Ctrl" %
% Rung: 2 %
% REJECT PUSHER START-STOP LOGIC %
SOR XIC B3:0/12 BST XIC B3:1/2 NXB XIC B3:0/5 XIO B3:1/3 BND OTE B3:0/5 EOR
%   B3:0/12  "System_Status 0 = System Off 1 = System Running" %
%   B3:1/2  "RejectPusher_Trig_Ct rl" %
%   B3:0/5  "Reject_PusherOut_ Ctrl" %
%   B3:1/3  "RejectPusher_Intrpt_ Ctrl" %
% Rung: 3 %
% OUTFEED CONVEYOR START-STOP LOGIC %
SOR XIC B3:0/12 BST XIC B3:1/4 NXB XIC B3:0/6 XIO B3:1/5 BND OTE B3:0/6 EOR
%   B3:0/12  "System_Status 0 = System Off 1 = System Running" %
%   B3:1/4  "OutfeedConv_Trig_C trl" %
%   B3:0/6  "OutfeedConvOut_Ctrl" %
%   B3:1/5  "OutfeedConv_Intrpt_C trl" %
% Rung: 4 %
% FILL VALVE START-STOP LOGIC %
SOR XIC B3:0/12 BST XIC B3:1/6 NXB XIC B3:0/3 XIO B3:1/7 BND OTE B3:0/3 EOR
%   B3:0/12  "System_Status 0 = System Off 1 = System Running" %
%   B3:1/6  "FillValve_Trig_ Ctrl" %
%   B3:0/3  "FillValve_Out_Ctrl" %
%   B3:1/7  "FillValve_Intrpt_Ctr l" %
% Rung: 5 %
SOR END EOR

LADDER 8 "CYCLE RST"
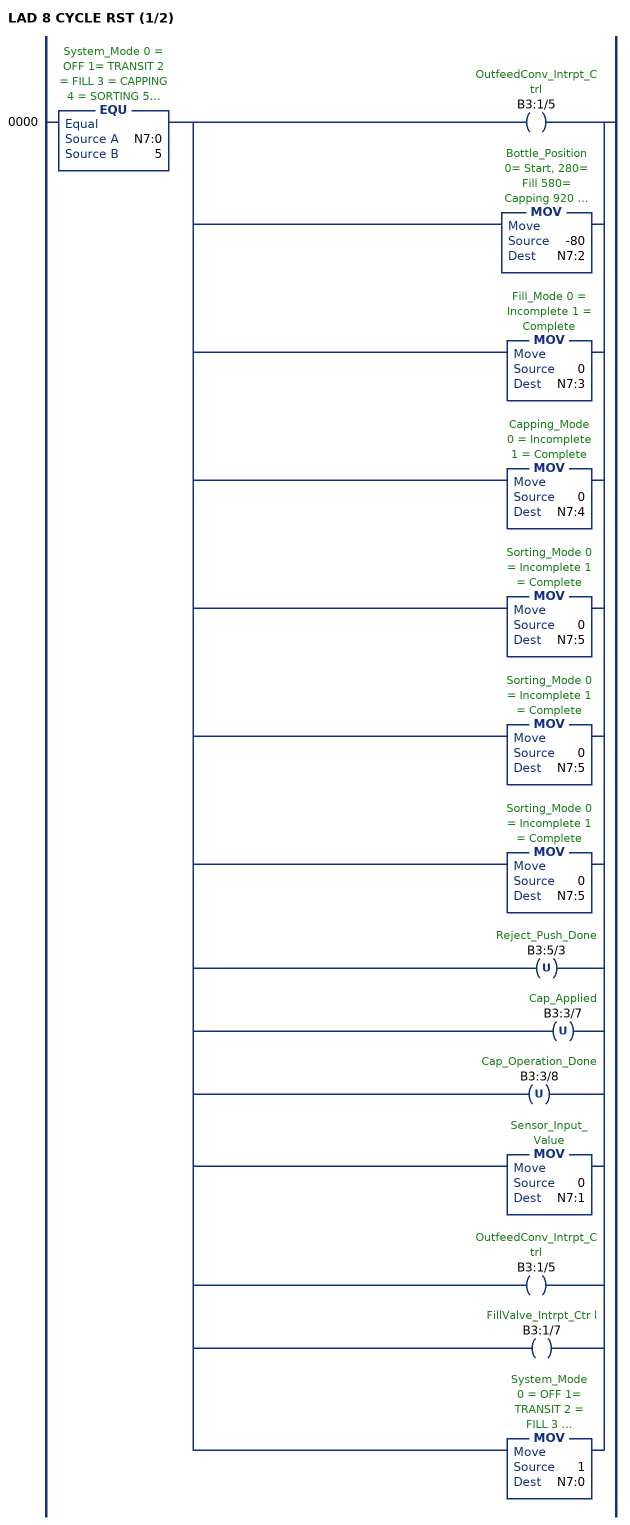
% Rung: 0 %
SOR EQU N7:0 5 BST OTE B3:1/5 NXB MOV -80 N7:2 NXB MOV 0 N7:3 NXB MOV 0 N7:4 NXB MOV 0 N7:5 NXB MOV 0 N7:5 NXB MOV 0 N7:5 NXB OTU B3:5/3 NXB OTU B3:3/7 NXB OTU B3:3/8 NXB MOV 0 N7:1 NXB OTE B3:1/5 NXB OTE B3:1/7 NXB MOV 1 N7:0 BND EOR
%   N7:0  "System_Mode 0 = OFF 1= TRANSIT 2 = FILL 3 = CAPPING 4 = SORTING 5= CYC.R" %
%   B3:1/5  "OutfeedConv_Intrpt_C trl" %
%   N7:2  "Bottle_Position 0= Start, 280= Fill 580= Capping 920 = Sorting" %
%   N7:3  "Fill_Mode 0 = Incomplete 1 = Complete" %
%   N7:4  "Capping_Mode 0 = Incomplete 1 = Complete" %
%   N7:5  "Sorting_Mode 0 = Incomplete 1 = Complete" %
%   B3:5/3  "Reject_Push_Done" %
%   B3:3/7  "Cap_Applied" %
%   B3:3/8  "Cap_Operation_Done" %
%   N7:1  "Sensor_Input_Value" %
%   B3:1/7  "FillValve_Intrpt_Ctr l" %

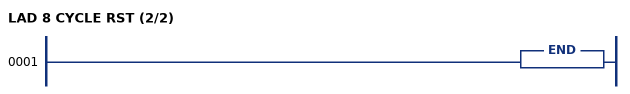
% Rung: 1 %
SOR END EOR

LADDER 9 "HOURMETER"
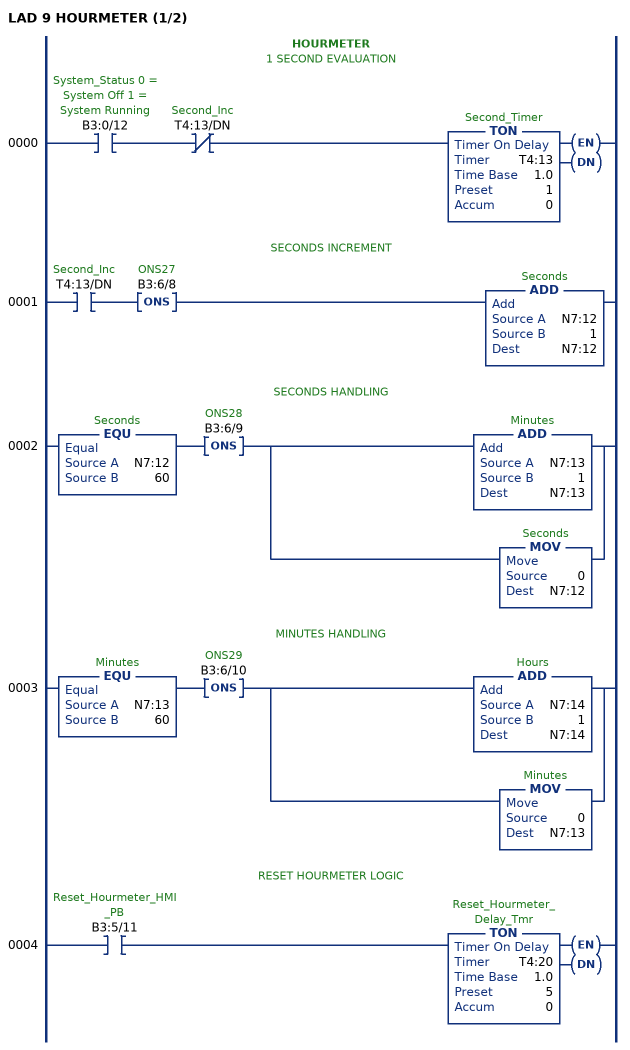
% Rung: 0 %
% TITLE: HOURMETER %
% 1 SECOND EVALUATION %
SOR XIC B3:0/12 XIO T4:13/DN TON T4:13 1.0 1 0 EOR
%   B3:0/12  "System_Status 0 = System Off 1 = System Running" %
%   T4:13/DN  "Second_Inc" %
%   T4:13  "Second_Timer" %
% Rung: 1 %
% SECONDS INCREMENT %
SOR XIC T4:13/DN ONS B3:6/8 ADD N7:12 1 N7:12 EOR
%   T4:13/DN  "Second_Inc" %
%   B3:6/8  "ONS27" %
%   N7:12  "Seconds" %
% Rung: 2 %
% SECONDS HANDLING %
SOR EQU N7:12 60 ONS B3:6/9 BST ADD N7:13 1 N7:13 NXB MOV 0 N7:12 BND EOR
%   N7:12  "Seconds" %
%   B3:6/9  "ONS28" %
%   N7:13  "Minutes" %
% Rung: 3 %
% MINUTES HANDLING %
SOR EQU N7:13 60 ONS B3:6/10 BST ADD N7:14 1 N7:14 NXB MOV 0 N7:13 BND EOR
%   N7:13  "Minutes" %
%   B3:6/10  "ONS29" %
%   N7:14  "Hours" %
% Rung: 4 %
% RESET HOURMETER LOGIC %
SOR XIC B3:5/11 TON T4:20 1.0 5 0 EOR
%   B3:5/11  "Reset_Hourmeter_HMI _PB" %
%   T4:20  "Reset_Hourmeter_ Delay_Tmr" %

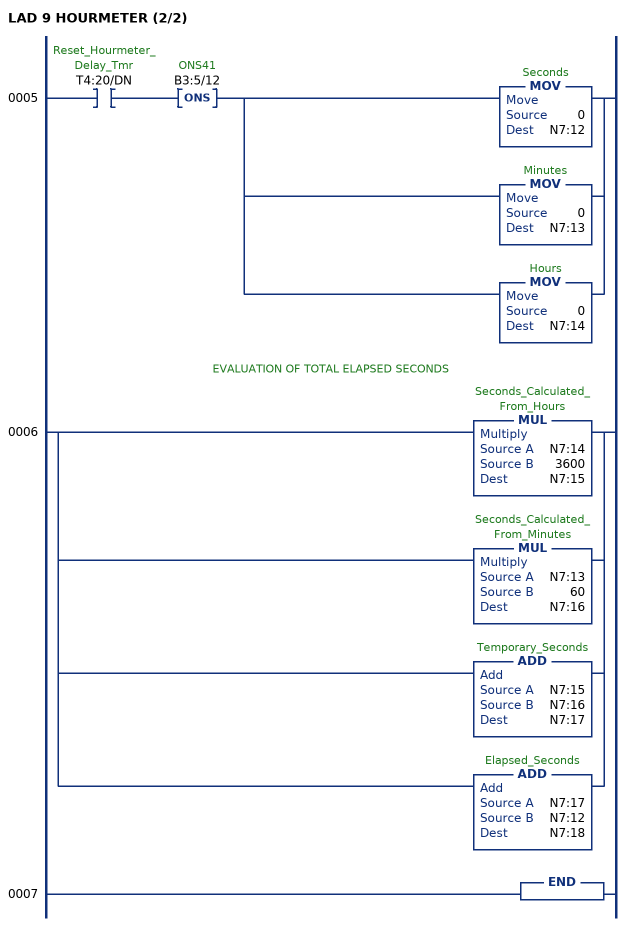
% Rung: 5 %
SOR XIC T4:20/DN ONS B3:5/12 BST MOV 0 N7:12 NXB MOV 0 N7:13 NXB MOV 0 N7:14 BND EOR
%   T4:20  "Reset_Hourmeter_ Delay_Tmr" %
%   B3:5/12  "ONS41" %
%   N7:12  "Seconds" %
%   N7:13  "Minutes" %
%   N7:14  "Hours" %
% Rung: 6 %
% EVALUATION OF TOTAL ELAPSED SECONDS %
SOR BST MUL N7:14 3600 N7:15 NXB MUL N7:13 60 N7:16 NXB ADD N7:15 N7:16 N7:17 NXB ADD N7:17 N7:12 N7:18 BND EOR
%   N7:14  "Hours" %
%   N7:15  "Seconds_Calculated_ From_Hours" %
%   N7:13  "Minutes" %
%   N7:16  "Seconds_Calculated_ From_Minutes" %
%   N7:17  "Temporary_Seconds" %
%   N7:12  "Seconds" %
%   N7:18  "Elapsed_Seconds" %
% Rung: 7 %
SOR END EOR

LADDER 10 "ALARMS"
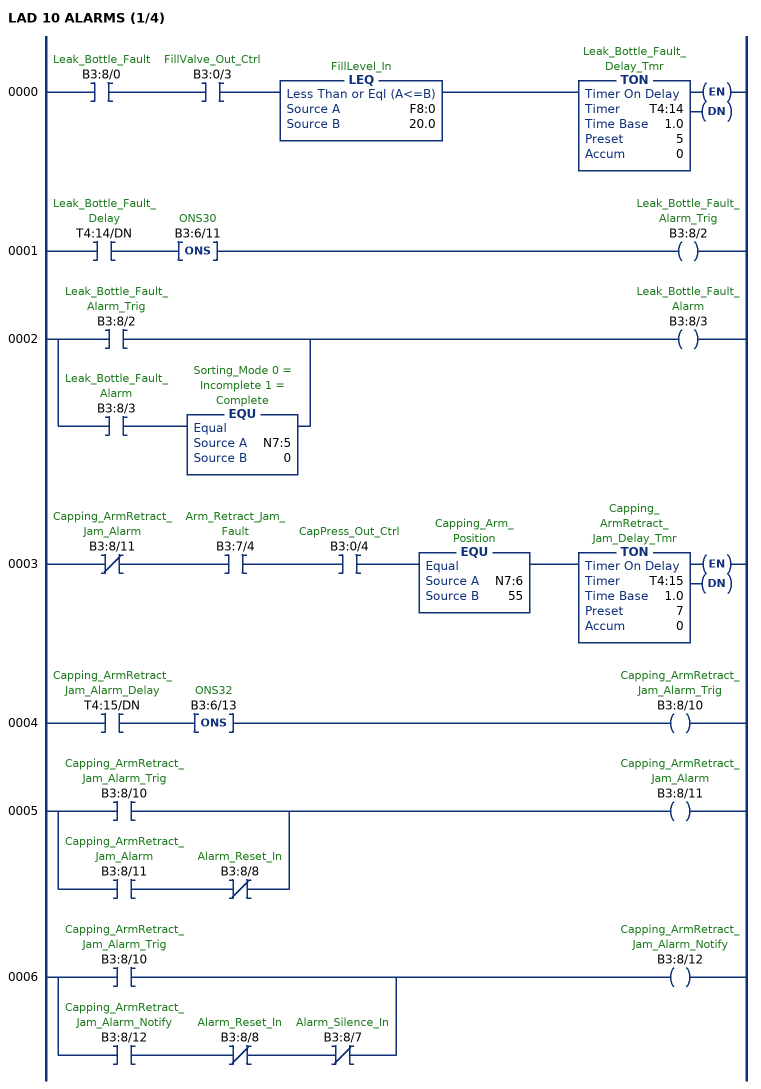
% Rung: 0 %
SOR XIC B3:8/0 XIC B3:0/3 LEQ F8:0 20.0 TON T4:14 1.0 5 0 EOR
%   B3:8/0  "Leak_Bottle_Fault" %
%   B3:0/3  "FillValve_Out_Ctrl" %
%   F8:0  "FillLevel_In" %
%   T4:14  "Leak_Bottle_Fault_ Delay_Tmr" %
% Rung: 1 %
SOR XIC T4:14/DN ONS B3:6/11 OTE B3:8/2 EOR
%   T4:14/DN  "Leak_Bottle_Fault_ Delay" %
%   B3:6/11  "ONS30" %
%   B3:8/2  "Leak_Bottle_Fault_ Alarm_Trig" %
% Rung: 2 %
SOR BST XIC B3:8/2 NXB XIC B3:8/3 EQU N7:5 0 BND OTE B3:8/3 EOR
%   B3:8/2  "Leak_Bottle_Fault_ Alarm_Trig" %
%   B3:8/3  "Leak_Bottle_Fault_ Alarm" %
%   N7:5  "Sorting_Mode 0 = Incomplete 1 = Complete" %
% Rung: 3 %
SOR XIO B3:8/11 XIC B3:7/4 XIC B3:0/4 EQU N7:6 55 TON T4:15 1.0 7 0 EOR
%   B3:8/11  "Capping_ArmRetract_ Jam_Alarm" %
%   B3:7/4  "Arm_Retract_Jam_ Fault" %
%   B3:0/4  "CapPress_Out_Ctrl" %
%   N7:6  "Capping_Arm_Position" %
%   T4:15  "Capping_ArmRetract_ Jam_Delay_Tmr" %
% Rung: 4 %
SOR XIC T4:15/DN ONS B3:6/13 OTE B3:8/10 EOR
%   T4:15/DN  "Capping_ArmRetract_ Jam_Alarm_Delay" %
%   B3:6/13  "ONS32" %
%   B3:8/10  "Capping_ArmRetract_ Jam_Alarm_Trig" %
% Rung: 5 %
SOR BST XIC B3:8/10 NXB XIC B3:8/11 XIO B3:8/8 BND OTE B3:8/11 EOR
%   B3:8/10  "Capping_ArmRetract_ Jam_Alarm_Trig" %
%   B3:8/11  "Capping_ArmRetract_ Jam_Alarm" %
%   B3:8/8  "Alarm_Reset_In" %
% Rung: 6 %
SOR BST XIC B3:8/10 NXB XIC B3:8/12 XIO B3:8/8 XIO B3:8/7 BND OTE B3:8/12 EOR
%   B3:8/10  "Capping_ArmRetract_ Jam_Alarm_Trig" %
%   B3:8/12  "Capping_ArmRetract_ Jam_Alarm_Notify" %
%   B3:8/8  "Alarm_Reset_In" %
%   B3:8/7  "Alarm_Silence_In" %

